PROGRAM MAIN
VAR
END_VAR

END_PROGRAM

(* stored: Version 1.1.0.1
   POU MAIN: Id {ac1bfdff-d286-48d9-b06e-2fe1fa515cf2} *)
